PROGRAM MAIN
VAR
	
	
END_VAR
VAR_OUTPUT
END_VAR


fbAct1();

END_PROGRAM

(* stored: Version 1.1.0.1, ProductVersion 3.1.4020.6
   POU MAIN: Id {88565b10-f526-4ac4-9c9a-5fc4dafa25eb}, SpecialFunc None *)
